Fanuc KAREL source: wspeed.kl

PROGRAM wspeed
%NOLOCKGROUP
VAR
  p : POSITION
  q : POSITION
  i : INTEGER
  r : REAL
BEGIN
  WITH $SPEED = 500 MOVE TO p
END wspeed
